// Mitsubishi GX Works2 project: EXC2V11   PLC: FX3G

// global labels: Global1
VAR_GLOBAL
  START_WORK_DAY AT X007 : BOOL;
  SYSTEM_ACTIVE_LED AT Y007 : BOOL;
  EMERGENCY_STOP AT X005 : BOOL;
  FAULT_LOW_STOCK AT M0 : BOOL;
  INIT_CYCLE_START AT X001 : BOOL;
  TYPE_REGULAR AT M10 : BOOL;
  TYPE_DELUXE AT M11 : BOOL;
  SAMPLED_TYPE_VALUE AT D200 : REAL;
  STOCK_RASPBERRY AT D0 : REAL;
  STOCK_LEMON AT D10 : REAL;
  STOCK_STABILIZER AT D2000 : REAL;
  STOCK_GUMMY_BEARS AT D30 : REAL;
  LED_STAGE_PREP AT Y000 : BOOL;
  COOLING_START AT X002 : BOOL;
  LED_STAGE_COOLING AT Y002 : BOOL;
  TEMP_SENSOR_10C AT X003 : BOOL;
  COOLING_TIMER AT TS1 : BOOL;
  MIXING_TIMER AT TS2 : BOOL;
  MIXING_REGULAR_ACTIVE AT M12 : BOOL;
  FLICKER_CLOCK_TIMER AT TS3 : BOOL;
  BLINK_TIMER_ELAPSED AT D300 : REAL;
  MIXING_LED_A AT Y005 : BOOL;
  MIXING_LED_B AT Y006 : BOOL;
  TOTAL_PACKS_STOCKED AT D110 : REAL;
  PREP_TIMER AT TS0 : BOOL;
  MIXING_DELUXE_ACTIVE AT M13 : BOOL;
  MIXING_TIMER_DELUXE AT TS3 : BOOL;
  MIXING_TIMER_REGULAR AT TS2 : BOOL;
  TOTAL_Current_PACKS_STOCKED AT D1110 : REAL;
  TOTAL_Previous_PACKS_STOCKED AT D1220 : REAL;
  New_Pack_Trigger AT M20 : BOOL;
  TOTAL_UNITS_STOCKED AT D180 : REAL;
  GUMMY_TYPE_INPUT AT D8280 : INT;
  FINAL_OUTPUT_RESULT AT D8282 : INT;
END_VAR

// task Task_01 (event TRUE, interval 0, priority 31): POU_01

PROGRAM POU_01
VAR
  TIMER_PREP : BOOL;
  TN0 : BOOL;
END_VAR
(* structured ladder/FBD written out as ST: instructions are called as NAME(EN, inputs, outputs); _pN, _eN, _tN stand for wires *)
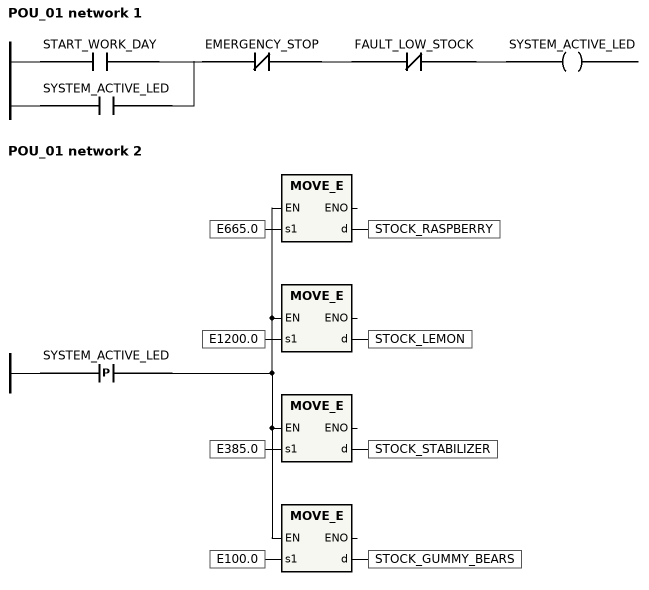
(* network 1 *)
SYSTEM_ACTIVE_LED := ((START_WORK_DAY OR SYSTEM_ACTIVE_LED) AND NOT EMERGENCY_STOP) AND NOT FAULT_LOW_STOCK;
(* network 2 *)
_p1 := LDP(TRUE, SYSTEM_ACTIVE_LED);
MOVE_E(_p1, E665.0, STOCK_RASPBERRY);
MOVE_E(_p1, E1200.0, STOCK_LEMON);
MOVE_E(_p1, E385.0, STOCK_STABILIZER);
MOVE_E(_p1, E100.0, STOCK_GUMMY_BEARS);
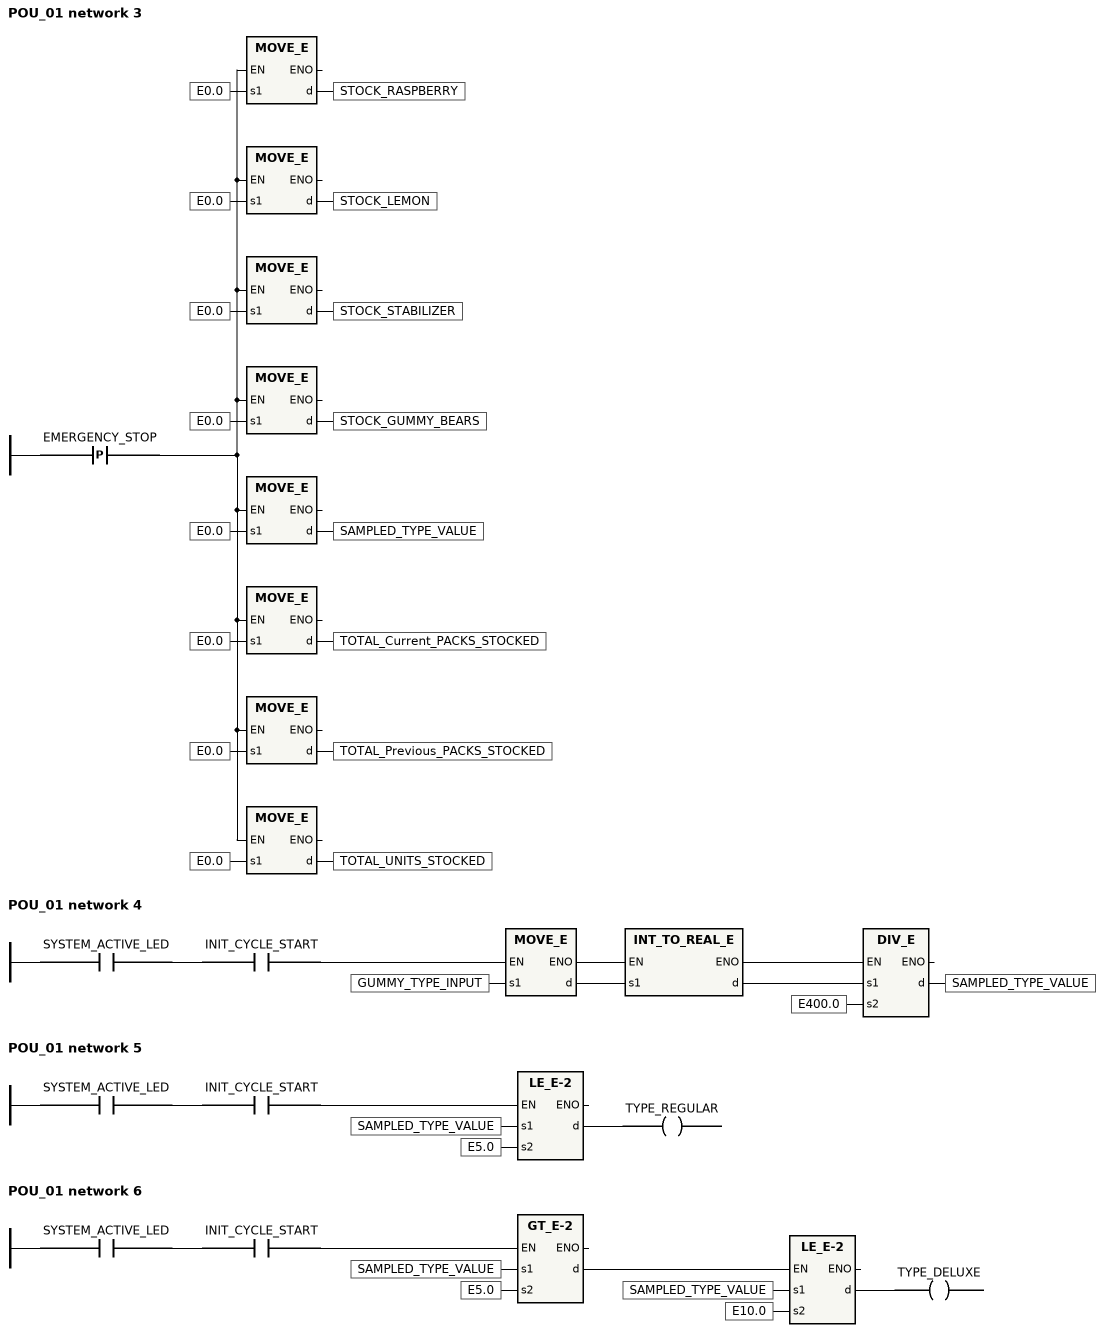
(* network 3 *)
_p1 := LDP(TRUE, EMERGENCY_STOP);
MOVE_E(_p1, E0.0, STOCK_RASPBERRY);
MOVE_E(_p1, E0.0, STOCK_LEMON);
MOVE_E(_p1, E0.0, STOCK_STABILIZER);
MOVE_E(_p1, E0.0, STOCK_GUMMY_BEARS);
MOVE_E(_p1, E0.0, SAMPLED_TYPE_VALUE);
MOVE_E(_p1, E0.0, TOTAL_Current_PACKS_STOCKED);
MOVE_E(_p1, E0.0, TOTAL_Previous_PACKS_STOCKED);
MOVE_E(_p1, E0.0, TOTAL_UNITS_STOCKED);
(* network 4 *)
_e2 := MOVE_E(SYSTEM_ACTIVE_LED AND INIT_CYCLE_START, GUMMY_TYPE_INPUT, _t1);
_e4 := INT_TO_REAL_E(_e2, _t1, _t3);
DIV_E(_e4, _t3, E400.0, SAMPLED_TYPE_VALUE);
(* network 5 *)
LE_E(SYSTEM_ACTIVE_LED AND INIT_CYCLE_START, SAMPLED_TYPE_VALUE, E5.0, _t1);
TYPE_REGULAR := _t1;
(* network 6 *)
GT_E(SYSTEM_ACTIVE_LED AND INIT_CYCLE_START, SAMPLED_TYPE_VALUE, E5.0, _t1);
LE_E(_t1, SAMPLED_TYPE_VALUE, E10.0, _t2);
TYPE_DELUXE := _t2;
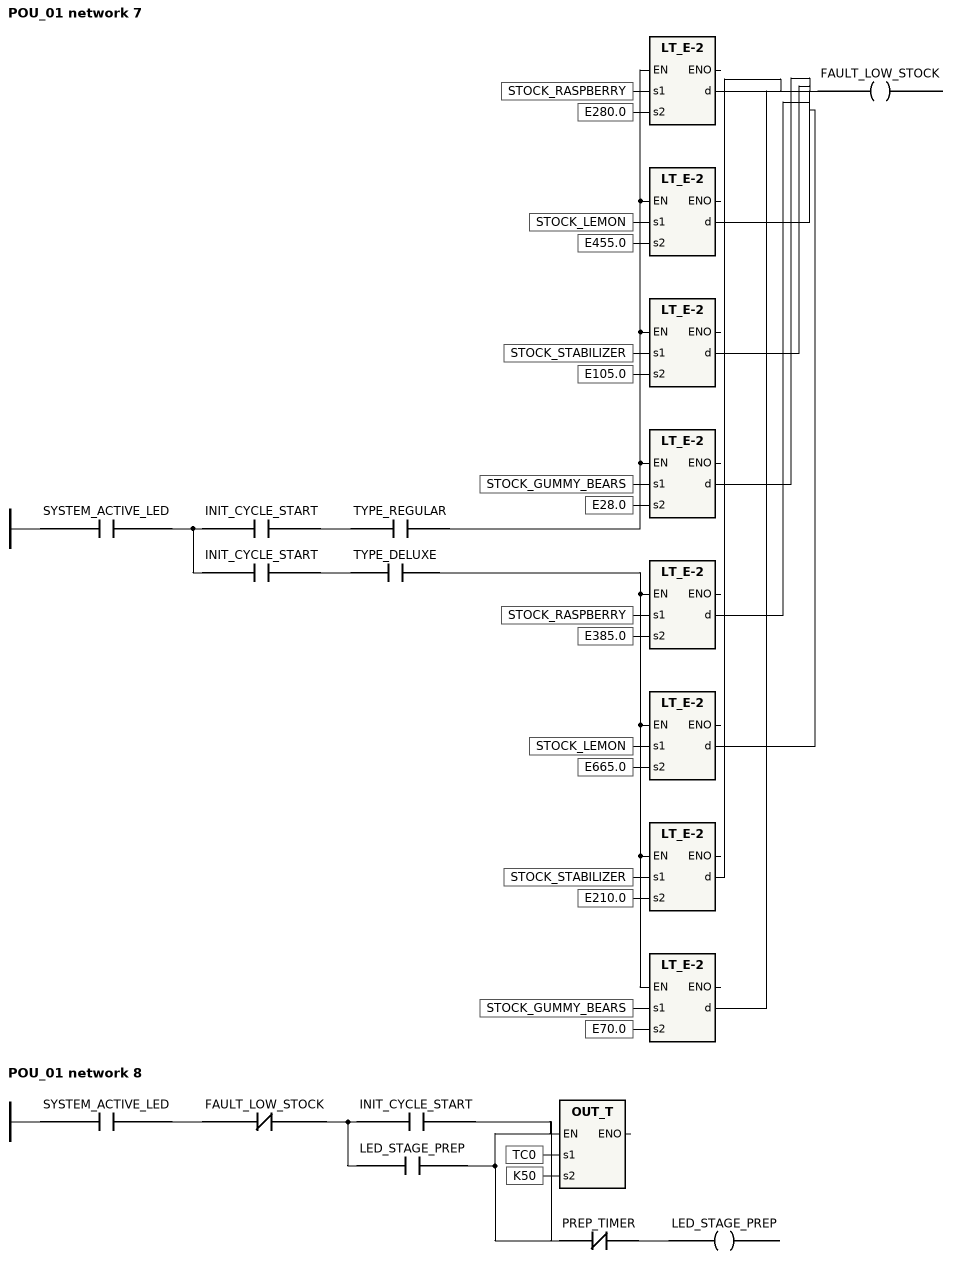
(* network 7 *)
_p1 := SYSTEM_ACTIVE_LED AND INIT_CYCLE_START AND TYPE_REGULAR;
LT_E(_p1, STOCK_RASPBERRY, E280.0, _t2);
LT_E(_p1, STOCK_LEMON, E455.0, _t3);
LT_E(_p1, STOCK_STABILIZER, E105.0, _t4);
LT_E(_p1, STOCK_GUMMY_BEARS, E28.0, _t5);
_p6 := SYSTEM_ACTIVE_LED AND INIT_CYCLE_START AND TYPE_DELUXE;
LT_E(_p6, STOCK_RASPBERRY, E385.0, _t7);
LT_E(_p6, STOCK_LEMON, E665.0, _t8);
LT_E(_p6, STOCK_STABILIZER, E210.0, _t9);
LT_E(_p6, STOCK_GUMMY_BEARS, E70.0, _t10);
FAULT_LOW_STOCK := _t2 OR _t3 OR _t4 OR _t5 OR _t7 OR _t8 OR _t9 OR _t10;
(* network 8 *)
_p1 := SYSTEM_ACTIVE_LED AND NOT FAULT_LOW_STOCK;
_p2 := (_p1 AND INIT_CYCLE_START) OR (_p1 AND LED_STAGE_PREP);
LED_STAGE_PREP := _p2 AND NOT PREP_TIMER;
OUT_T(_p2, TC0, K50);
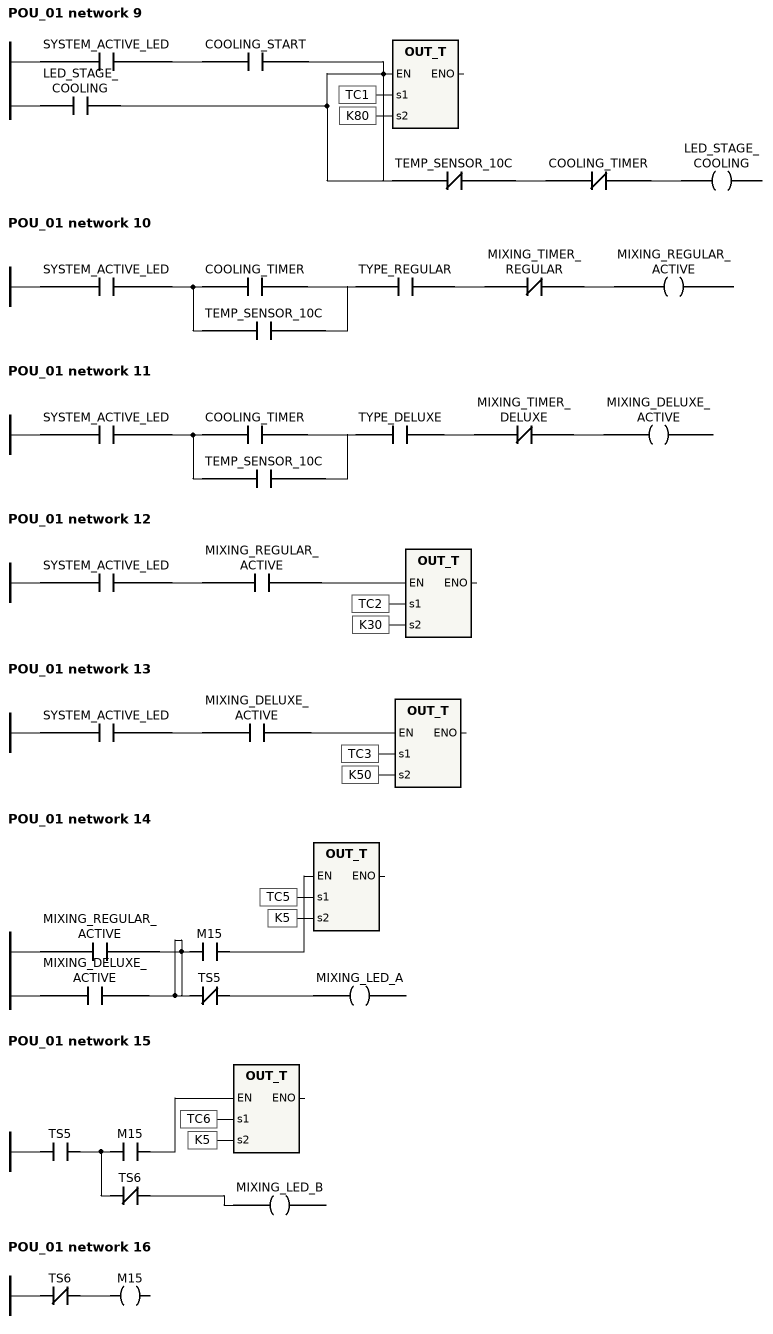
(* network 9 *)
_p1 := (SYSTEM_ACTIVE_LED AND COOLING_START) OR LED_STAGE_COOLING;
LED_STAGE_COOLING := _p1 AND NOT TEMP_SENSOR_10C AND NOT COOLING_TIMER;
OUT_T(_p1, TC1, K80);
(* network 10 *)
MIXING_REGULAR_ACTIVE := (((SYSTEM_ACTIVE_LED AND COOLING_TIMER) OR (SYSTEM_ACTIVE_LED AND TEMP_SENSOR_10C)) AND TYPE_REGULAR) AND NOT MIXING_TIMER_REGULAR;
(* network 11 *)
MIXING_DELUXE_ACTIVE := (((SYSTEM_ACTIVE_LED AND COOLING_TIMER) OR (SYSTEM_ACTIVE_LED AND TEMP_SENSOR_10C)) AND TYPE_DELUXE) AND NOT MIXING_TIMER_DELUXE;
(* network 12 *)
OUT_T(SYSTEM_ACTIVE_LED AND MIXING_REGULAR_ACTIVE, TC2, K30);
(* network 13 *)
OUT_T(SYSTEM_ACTIVE_LED AND MIXING_DELUXE_ACTIVE, TC3, K50);
(* network 14 *)
_p1 := MIXING_REGULAR_ACTIVE OR MIXING_DELUXE_ACTIVE;
OUT_T(_p1 AND M15, TC5, K5);
MIXING_LED_A := _p1 AND NOT TS5;
(* network 15 *)
OUT_T(TS5 AND M15, TC6, K5);
MIXING_LED_B := TS5 AND NOT TS6;
(* network 16 *)
M15 := NOT TS6;
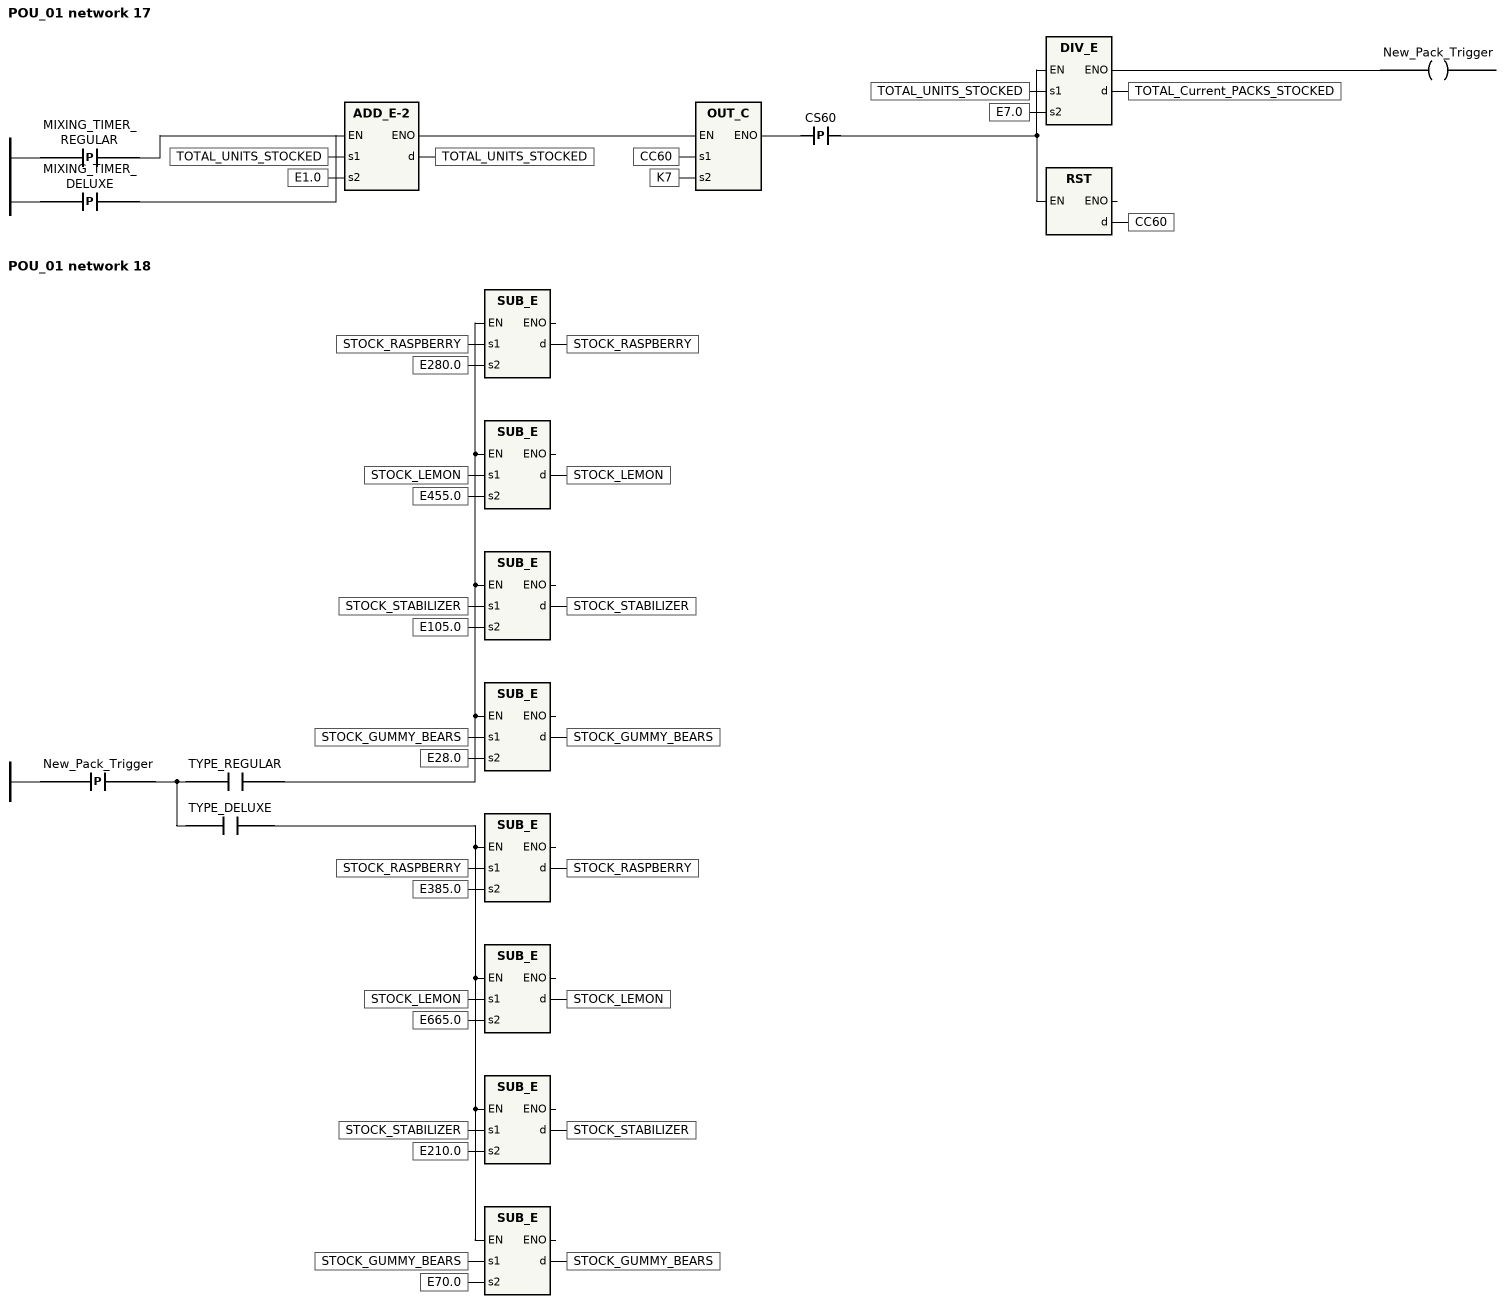
(* network 17 *)
_e1 := ADD_E(LDP(TRUE, MIXING_TIMER_REGULAR) OR LDP(TRUE, MIXING_TIMER_DELUXE), TOTAL_UNITS_STOCKED, E1.0, TOTAL_UNITS_STOCKED);
_e2 := OUT_C(_e1, CC60, K7);
_p3 := _e2 AND LDP(TRUE, CS60);
_e4 := DIV_E(_p3, TOTAL_UNITS_STOCKED, E7.0, TOTAL_Current_PACKS_STOCKED);
New_Pack_Trigger := _e4;
RST(_p3, CC60);
(* network 18 *)
_p1 := LDP(TRUE, New_Pack_Trigger);
_p2 := _p1 AND TYPE_REGULAR;
SUB_E(_p2, STOCK_RASPBERRY, E280.0, STOCK_RASPBERRY);
SUB_E(_p2, STOCK_LEMON, E455.0, STOCK_LEMON);
SUB_E(_p2, STOCK_STABILIZER, E105.0, STOCK_STABILIZER);
SUB_E(_p2, STOCK_GUMMY_BEARS, E28.0, STOCK_GUMMY_BEARS);
_p3 := _p1 AND TYPE_DELUXE;
SUB_E(_p3, STOCK_RASPBERRY, E385.0, STOCK_RASPBERRY);
SUB_E(_p3, STOCK_LEMON, E665.0, STOCK_LEMON);
SUB_E(_p3, STOCK_STABILIZER, E210.0, STOCK_STABILIZER);
SUB_E(_p3, STOCK_GUMMY_BEARS, E70.0, STOCK_GUMMY_BEARS);
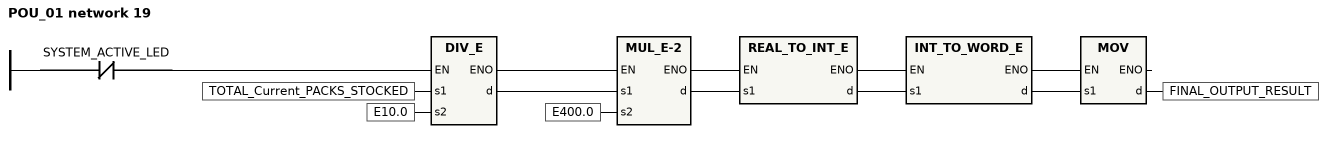
(* network 19 *)
_e2 := DIV_E(NOT SYSTEM_ACTIVE_LED, TOTAL_Current_PACKS_STOCKED, E10.0, _t1);
_e4 := MUL_E(_e2, _t1, E400.0, _t3);
_e6 := REAL_TO_INT_E(_e4, _t3, _t5);
_e8 := INT_TO_WORD_E(_e6, _t5, _t7);
MOV(_e8, _t7, FINAL_OUTPUT_RESULT);
END_PROGRAM
